# EPICS alarm handler configuration: mps_database/bare/alarms/areas/mpln_ltus_mp06.alhConfig
GROUP NULL MPLN:LTUS:MP06:1
$ALIAS MPS Link Node 209
$GUIDANCE
LTUH MPS
   Group Name: MPLN:LTUS:MP06:1
   Summary PV:  MPLN:LTUS:MP06:1:STATSUMY
$END
CHANNEL  MPLN:LTUS:MP06:1    MPLN:LTUS:MP06:1:MPS_EN_RBV		-----
CHANNEL  MPLN:LTUS:MP06:1    MPLN:LTUS:MP06:1:LC1_MODE_RBV		-----
